TYPE ST_TestDefinition :
	STRUCT
		TestId : T_MaxString;
		Status : E_TestStatus;
	END_STRUCT
END_TYPE

(* stored: Version 1.1.0.1
   DUT ST_TestDefinition: Id {e631d038-4e4a-4dc0-a404-8a4a12f8f78f} *)
